// TIA Portal V21 export
DATA_BLOCK "DoDb"   // DB109
// stored: AutoNumber false, InstanceOfName DoFb, InstanceOfType FB
"DoFb"
   // VAR_INPUT
   //    sec : Bool;
   //    AlarmAck : Bool;
   //    AlwaysTrue : Bool;
   //    AlwaysFalse : Bool;
   //    Interlock : Bool;
   // END_VAR
   // VAR
   //    Do01 { S7_SetPoint := 'True'} : "DigitalOutput";
   //    Do02 { S7_SetPoint := 'True'} : "DigitalOutput";
   //    Do03 { S7_SetPoint := 'True'} : "DigitalOutput";
   //    Do04 { S7_SetPoint := 'True'} : "DigitalOutput";
   //    Do05 { S7_SetPoint := 'True'} : "DigitalOutput";
   //    Do06 { S7_SetPoint := 'True'} : "DigitalOutput";
   //    Do07 { S7_SetPoint := 'True'} : "DigitalOutput";
   //    Do08 { S7_SetPoint := 'True'} : "DigitalOutput";
   //    Do09 { S7_SetPoint := 'True'} : "DigitalOutput";
   //    Do10 { S7_SetPoint := 'True'} : "DigitalOutput";
   // END_VAR
BEGIN
END_DATA_BLOCK
